Staubli VAL3: oResetFault.pgx

public program oResetFault()
// Reseta rele de seguranca
begin
  dioSet(oResetFault,1)
  delay(1)
  dioSet(oResetFault,0)
end
